Staubli VAL3: remGetnGlobal.pgx

program remGetnGlobal(num& nGlobal[] (dimensions=1), string& sCmd[] (dimensions=1), string& sReturn[] (dimensions=1))
begin
  // Get an arbitrary global value and return it
  //
  logMsg("call remGetnGlobal")
  sReturn=sCmd+" "+toString(sNumConv,nGlobal)
end
